// TIA Portal V20 export
// export: Created 2025-12-01T14:56:59.4390945Z, ExportSetting None, DisplayName Totally Integrated Automation Portal, DisplayVersion V20 Update 3, DisplayName TIA Portal Openness, DisplayVersion V20 Update 3, DisplayName TIA Portal Version Control Interface, DisplayVersion V20 Update 3, DisplayName STEP 7 Professional, DisplayVersion V20 Update 3, DisplayName STEP 7 Safety, DisplayVersion V20 Update 2, DisplayName WinCC Basic/Comfort/Advanced, DisplayVersion V20 Update 3, DisplayName WinCC Professional, DisplayVersion V20 Update 3, DisplayName WinCC Unified, DisplayVersion V20 Update 3
FUNCTION "FC410_Calc_Posicion_Relativa" : Void   // FC410, LAD
TITLE = Calculo de la posion relativa.
{ S7_Optimized_Access := 'FALSE' }
// Esta FC lo que hace es calcular la posicion relativa, respecto a un "0" que no es cero. Es decir, el enconder pasara por un sensor de homming, pero el valor del encoder seguira contando hacia adelante. Por lo que al pasar por el homming, nos tendremos que guardar esa informacion para que sea utilizada en el ciclo actual. Tenemos solo una nota que hacer, el encoder tiene un numero maximo, despues de alcanzado este numero, la cuenta inicia otra vez en 0. Por lo que tenemos que calcular siempre por abajo de este valor maximo. Para que el programa no compare con valores superiores a este valor maximo
// stored: AutoNumber false, SetENOAutomatically false
   VAR_INPUT
      Pos_Absoluta : DInt;
      Mem_Encoder_Home : DInt;
      Lim_Superior_Encoder : DInt;
   END_VAR
   VAR_OUTPUT
      Pos_Relativa : DInt;
      Pos_Mayor_que_max : Bool;
   END_VAR
   VAR_TEMP
      comp_pos_soltar_carga : DInt;
   END_VAR
BEGIN

NETWORK
TITLE = 


      L     #Pos_Absoluta;
      L     #Mem_Encoder_Home;
      +D;
      T     #comp_pos_soltar_carga;

//si la suma es mayor que el limite superior encoder entonces
//restarle el lim_sup_encoder a la cantidad resultante
      L     #comp_pos_soltar_carga;
      L     #Lim_Superior_Encoder;
      >D;
      JCN   mesc;


//cantidad es mayor
      L     #Pos_Absoluta;
      L     #Mem_Encoder_Home;
      +D;
      L     #Lim_Superior_Encoder;
      -D;
      T     #Pos_Relativa;

//ponemos una marca a 1, para saber que es mayor
      S     #Pos_Mayor_que_max;
      JU    fina;


mesc: NOP   0;
//cantidad menor
      L     #Pos_Absoluta;
      L     #Mem_Encoder_Home;
      +D;
      T     #Pos_Relativa;
//reseteamos la marca
      R     #Pos_Mayor_que_max;
fina: NOP   0;








END_FUNCTION
